# B&R Automation Studio project TestOpcUaServer
Automation Studio 6.5.2.12; technology packages: OpcUaCs 6.6.1

## Configuration Sim

CPU PC_any, AutomationRuntime 6.6.2, Build 11.3.0

### Task classes (Cpu.sw)
```
Cyclic#1:
  Program <- Program.prg
Binaries: udbdef, FWRules, TCData, sysconf, User, iomap, ashwd, BRRole, asfw, arconfig, ashwac, UaCsConfig
Libraries: runtime, UaCore, AsIecCon
```

### Hardware
```
PC : PC_any v1.1.2.0 (OrderNumber=PC)
  FileDevice1
  FileDeviceName1 = USER
  FileDevicePath1 = USER_PATH
```

## Logical view

### Global.typ - Global data types
```iecst
TYPE
	SimpleStruct : 	STRUCT
		xData1 : BOOL;
		xData2 : BOOL;
		xData3 : BOOL;
		xData4 : BOOL;
		iData1 : INT;
		iData2 : INT;
		iData3 : INT;
		iData4 : INT;
	END_STRUCT;
END_TYPE
```

### Global.var - Global variables
```iecst
VAR
	SimpleStruct_1 : SimpleStruct;
END_VAR
```

### Program Logical/Program (IEC)

#### Cyclic.st
```iecst
PROGRAM _CYCLIC
	(* Insert code here *)
	SimpleStruct_1;

END_PROGRAM
```

Listed in the project but not available here: Logical/Libraries
